TYPE M2PotentiometerAxisConfig :
STRUCT
	///Settings which are general for all axes
	general: M2AxisGeneralConfig;
	///Position = voltage * correctionFactor * voltageToPosition
	voltageCorrectionFactor: LREAL;
END_STRUCT
END_TYPE

(* stored: Version 1.1.0.1, ProductVersion 3.1.4019.2
   DUT M2PotentiometerAxisConfig: Id {7245fe30-3517-46b6-aece-163a7b4446e8} *)
